FUNCTION F_ReactorIndexToAnalogControllerIndex : UINT
VAR_INPUT
	i : UINT;
END_VAR
VAR
END_VAR

F_ReactorIndexToAnalogControllerIndex := i + GVL_CONSTANT.NumFlowController

END_FUNCTION

(* stored: Version 1.1.0.1, ProductVersion 3.1.4026.11
   POU F_ReactorIndexToAnalogControllerIndex: Id {e107827f-687c-44bb-b3b3-9f5c877a3adc}, SpecialFunc None *)
